FUNCTION_BLOCK FB_Cylinder
VAR_INPUT
	I_GoToHP 	:	BOOL;
	I_GoToWP 	:	BOOL;
	bSensorHP	:	BOOL;
	bSensorWP	:	BOOL;
	
END_VAR
VAR_OUTPUT
	Q_CoilToHP : BOOL;
	Q_CoilToWP : BOOL;
END_VAR
VAR
	bEnable			:	BOOL 	:= TRUE;
	bConfirmError	:	BOOL;

	bSensorWP_check	:	BOOL;
	bSensorHP_check	:	BOOL;
	Cmd_ToHP_act	:	BOOL;
	Cmd_ToWP_act	:	BOOL;

	TON_HP	:	TON;
	TON_WP	:	TON;
	timeHP	:	TIME := T#5S;
	timeWP	:	TIME := T#5S;
	
	iError	:	INT;
	sError	:	STRING;

END_VAR

ConfirmError();

IF bEnable  THEN
	TON_HP(IN := Cmd_ToHP_act, PT := timeHP);
	TON_WP(IN := Cmd_ToWP_act, PT := timeWP);

	CheckErrors();
END_IF

ACTION ConfirmError:
(*
IF SafetyIO.Common.Q_Safety_ErrorACK[1]  THEN
	Enable := TRUE;
END_IF
*)


IF bConfirmError THEN
	bEnable := TRUE;
	iError := 0;
	Cmd_ToHP_act := FALSE;
	Cmd_ToWP_act := FALSE;
	bConfirmError := FALSE;
END_IF
END_ACTION

ACTION GoToHP:
IF bEnable  THEN
	Q_CoilToHP 	:=	TRUE;
	Q_CoilToWP	:= 	FALSE;
	Cmd_ToHP_act:=	TRUE;
END_IF
END_ACTION

ACTION GoToWP:
IF bEnable  THEN
	Q_CoilToHP 	:=	FALSE;
	Q_CoilToWP	:= 	TRUE;
	Cmd_ToWP_act:=	TRUE;
END_IF
END_ACTION

ACTION CheckErrors:
IF bSensorWP THEN
	bSensorWP_check	:= TRUE;
ELSIF bSensorHP THEN
	bSensorHP_check	:= TRUE;
END_IF

//Control Errors for WP
IF TON_WP.Q AND NOT bSensorWP THEN
	IF bSensorWP_check THEN
		iError := 3;
		bSensorWP_check := FALSE;
	ELSE
		iError := 1;
	END_IF
	
//Control Errors for HP
ELSIF TON_HP.Q AND NOT bSensorHP THEN
	IF bSensorHP_check THEN
		iError := 4;
		bSensorHP_check := FALSE;
	ELSE
		iError := 2;
	END_IF
	
//Control for 'Both sensors error'
ELSIF
	bSensorHP AND bSensorWP THEN
	iError := 5;
END_IF

IF iError <> 0 THEN
	bEnable := FALSE;
END_IF

CASE iError OF
	0:	sError := 'OK';
	1:	sError := 'ERROR: Cylinder didnt reach WP on time';
	2:	sError := 'ERROR: Cylinder didnt reach HP on time';
	3:	sError := 'ERROR: Cylinder leaved HP';
	4:	sError := 'ERROR: Cylinder leaved WP';
	5:	sError := 'ERROR: Both sensors for HP and WP activated';
	
END_CASE
END_ACTION

END_FUNCTION_BLOCK

(* stored: Version 1.1.0.1, ProductVersion 3.1.4024.10
   POU FB_Cylinder: Id {5fa301b1-edb2-4339-85fb-9fd3cc3104f0}, SpecialFunc None
   Action ConfirmError: Id {b402ecb1-3ac3-4649-b2f9-79e8fba149b3}
   Action GoToHP: Id {4bdd60dd-625f-40b0-b4e3-c09a52daa24f}
   Action GoToWP: Id {4cbba615-8858-40b7-9864-872ec30fcd3f}
   Action CheckErrors: Id {a2444354-b0d2-44c3-bb0a-177409c7a92f} *)
